FUNCTION_BLOCK FB_Station
VAR_INPUT
	// Whole Station Init finished
	bInitFinished						: BOOL;
	
	// All E-Stop buttons
	EmergencyStop 						: BOOL;
	// From safety project
	SafetyReady 						: BOOL;
	// All door sensors
	Interlock 							: BOOL;
END_VAR
VAR_OUTPUT
	// Station Actual Status 
	diStationState 						: EN_StationStatus;
	
	// Stop executions
	bStop								: BOOL;
	
	// Reset Alarms
	 bAlarmReset						: BOOL;
END_VAR
VAR
	bStopButton 			AT %I* 		: BOOL;
	bStartButton 			AT %I* 		: BOOL;
	bResetButton			AT %I* 		: BOOL;

	bStopInterface 						: BOOL;
	bPauseInterface 					: BOOL;
	bInitStartInterface					: BOOL;
	bAutoStartInterface 				: BOOL;
	bResetInterface						: BOOL;
	OpUser 								: BOOL;

	AutoModeSelector 		AT %I* 		: BOOL;
	PressureSwitch 			AT %I* 		: BOOL;
	
	// Delay for stoppping machine with button 
	ton_stopMachineDelay 				: TON;
	
	// Delay for starts machine with button
	ton_startInitStartButtonDelay 		: TON;
END_VAR

StatusControl();
Alarm();

METHOD Alarm
VAR_INPUT
END_VAR
END_METHOD

METHOD StatusControl
VAR_INPUT
END_VAR

VAR
	// Safe operation condition in any mode
	bSafeOperationCondition			: BOOL;
	
	// Condtion for any Auto operation mode
	bAutoAvailable					: BOOL;
	
	// Condition for Maintenance operation mode
	bManualAvailable				: BOOL;
END_VAR
//	Condition for operate machine safely in any mode
	bSafeOperationCondition					:=	SafetyReady AND Interlock AND PressureSwitch;

//	Condition for operation in Auto Mode
	bAutoAvailable							:=	bSafeOperationCondition AND AutoModeSelector;

//	Condition for operation in Maintenance Mode
	bManualAvailable						:=	bSafeOperationCondition AND OpUser AND (NOT AutoModeSelector);
	
//	Stopping machine with button delay
	ton_stopMachineDelay(IN:=bStopButton,PT:=T#3S);
	
//	Starting machine with button delay
	ton_startInitStartButtonDelay(IN:=bStartButton,PT:=T#2S);
	
//	For controlling reset general output
	bAlarmReset								:=	bResetButton OR bResetInterface;
 
//	For controlling stop general output
	bStop									:=	bStopButton OR bStopInterface;

//	For Stopping the machine
	CASE diStationState OF
		EN_StationStatus.initializing :		// Initializing
			IF (NOT bAutoAvailable) OR bPauseInterface OR bStopInterface OR bStopButton THEN	
				diStationState				:=EN_StationStatus.stopped;
			END_IF;
		EN_StationStatus.idle :				//	Idle
			IF (NOT bAutoAvailable) OR (NOT bInitFinished) OR bStopInterface OR ton_stopMachineDelay.Q  THEN
				diStationState				:=EN_StationStatus.stopped;
			END_IF;
		EN_StationStatus.running:			// Running
			IF (NOT bAutoAvailable) OR (NOT bInitFinished) OR bStopInterface THEN
				diStationState				:=EN_StationStatus.stopped;
			END_IF;
		EN_StationStatus.maintenance:		// Maintenance
			IF (NOT bManualAvailable) THEN
				diStationState				:=EN_StationStatus.stopped;
			END_IF;
		EN_StationStatus.eStopped:			// E Stopped
			IF NOT EmergencyStop THEN
				diStationState				:=EN_StationStatus.stopped;
			END_IF;
	END_CASE;

//	For setting machine in Initialization or Running
	IF bAutoAvailable THEN
		CASE diStationState OF
			EN_StationStatus.stopped:		//	Stopped
				IF bInitStartInterface OR ton_startInitStartButtonDelay.Q THEN
					diStationState			:=EN_StationStatus.initializing;
				END_IF;
			EN_StationStatus.idle:			//	Idle
				IF bAutoStartInterface OR ton_startInitStartButtonDelay.Q THEN
					diStationState			:=EN_StationStatus.running;
				END_IF;
		END_CASE;
	END_IF;

//	For setting machine in Idle mode
	CASE diStationState OF
		EN_StationStatus.initializing:		// Initializing
			IF 	bInitFinished THEN
				diStationState				:=EN_StationStatus.idle;
			END_IF;
		EN_StationStatus.running:			// Running
			IF bStopButton OR bPauseInterface THEN
				diStationState				:=EN_StationStatus.idle;
			END_IF;
	END_CASE;

//	For setting machine in Maintenance mode
	IF bManualAvailable AND (diStationState=EN_StationStatus.stopped) THEN
		diStationState						:=EN_StationStatus.maintenance;
	END_IF;

//	For setting machine in E Stopped mode
	IF (EmergencyStop) AND (diStationState<>EN_StationStatus.eStopped) THEN
		diStationState						:=EN_StationStatus.eStopped;
	END_IF;
END_METHOD

END_FUNCTION_BLOCK

(* stored: Version 1.1.0.1, ProductVersion 3.1.4024.12
   POU FB_Station: Id {b1f4bc39-0056-4dd5-b97d-7e260e33bca2}, SpecialFunc None
   Method Alarm: Id {8d2e99f7-b30c-4f20-929c-ae47dd18aa97}
   Method StatusControl: Id {aa6b9823-9b73-4f62-a403-3df5fbc22a16} *)
